// TIA Portal V20 export
VAR_GLOBAL   // PLC tag table "Outputs"
   "Lamp 1 ON" AT %Q0.0 : Bool;
   "Lamp 2 ON" AT %Q0.1 : Bool;
   "Lamp 3 ON" AT %Q0.2 : Bool;
   "Lamp 4 ON" AT %Q0.3 : Bool;
   "Lamp 5 ON" AT %Q0.4 : Bool;
   "Lamp 6 ON" AT %Q0.5 : Bool;
   "Lamp 7 ON" AT %Q0.6 : Bool;
   "Lamp 8 ON" AT %Q0.7 : Bool;
   I_am_a_double_integer AT %QD1 : DInt;
END_VAR
